// TIA Portal V20 export
FUNCTION_BLOCK "Type_8"   // FB8, GRAPH
// stored: GraphVersion 2.0, SetENOAutomatically false
   // inherited from GRAPH_BASE
   VAR_INPUT
      OFF_SQ { ExternalAccessible := 'False'; ExternalVisible := 'False'; ExternalWritable := 'False'} : Bool := false;   // Turn sequence off
      INIT_SQ { ExternalAccessible := 'False'; ExternalVisible := 'False'; ExternalWritable := 'False'} : Bool := false;   // Set sequence to initial state
      ACK_EF { ExternalAccessible := 'False'; ExternalVisible := 'False'; ExternalWritable := 'False'} : Bool := false;   // Acknowledge all errors and faults
      S_PREV { ExternalAccessible := 'False'; ExternalVisible := 'False'; ExternalWritable := 'False'} : Bool := false;   // Output previous step in parameter S_NO
      S_NEXT { ExternalAccessible := 'False'; ExternalVisible := 'False'; ExternalWritable := 'False'} : Bool := false;   // Indicate next step in parameter S_NO
      SW_AUTO { ExternalAccessible := 'False'; ExternalVisible := 'False'; ExternalWritable := 'False'} : Bool := false;   // Automatic mode
      SW_TAP { ExternalAccessible := 'False'; ExternalVisible := 'False'; ExternalWritable := 'False'} : Bool := false;   // Semiautomatic/switch with transition
      SW_TOP { ExternalAccessible := 'False'; ExternalVisible := 'False'; ExternalWritable := 'False'} : Bool := false;   // Semiautomatic/ignore transition
      SW_MAN { ExternalAccessible := 'False'; ExternalVisible := 'False'; ExternalWritable := 'False'} : Bool := false;   // Manual mode
      S_SEL { ExternalAccessible := 'False'; ExternalVisible := 'False'; ExternalWritable := 'False'} : Int := 0;   // Select step to be output to S_NO
      S_ON { ExternalAccessible := 'False'; ExternalVisible := 'False'; ExternalWritable := 'False'} : Bool := false;   // Activate step indicated in S_NO
      S_OFF { ExternalAccessible := 'False'; ExternalVisible := 'False'; ExternalWritable := 'False'} : Bool := false;   // Disable step indicated in S_NO
      T_PUSH { ExternalAccessible := 'False'; ExternalVisible := 'False'; ExternalWritable := 'False'} : Bool := false;   // Enable transition to switch in semi automatic mode
   END_VAR
   VAR_OUTPUT
      S_NO { ExternalAccessible := 'False'; ExternalVisible := 'False'; ExternalWritable := 'False'} : Int := 0;   // Step number
      S_MORE { ExternalAccessible := 'False'; ExternalVisible := 'False'; ExternalWritable := 'False'} : Bool := false;   // More steps are available and can be shown in S_NO
      S_ACTIVE { ExternalAccessible := 'False'; ExternalVisible := 'False'; ExternalWritable := 'False'} : Bool := false;   // Step indicated in S_NO is active
      ERR_FLT { ExternalAccessible := 'False'; ExternalVisible := 'False'; ExternalWritable := 'False'} : Bool := false;   // Interlock or supervision group error
      AUTO_ON { ExternalAccessible := 'False'; ExternalVisible := 'False'; ExternalWritable := 'False'} : Bool := false;   // Automatic mode is active
      TAP_ON { ExternalAccessible := 'False'; ExternalVisible := 'False'; ExternalWritable := 'False'} : Bool := false;   // Semiautomatic mode/step with transition enabled
      TOP_ON { ExternalAccessible := 'False'; ExternalVisible := 'False'; ExternalWritable := 'False'} : Bool := false;   // Semiautomatic mode/ignore transition enabled
      MAN_ON { ExternalAccessible := 'False'; ExternalVisible := 'False'; ExternalWritable := 'False'} : Bool := false;   // Manual mode is active
   END_VAR
BEGIN
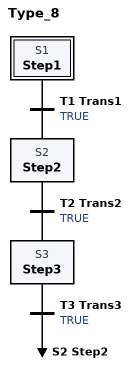
   // sequencer 1
   INITIAL_STEP Step1:   // S1, max time T#10S, warning time T#7S
   END_STEP
   TRANSITION Trans1 FROM Step1 TO Step2   // T1
      := TRUE;
   END_TRANSITION
   STEP Step2:   // S2, max time T#10S, warning time T#7S
   END_STEP
   TRANSITION Trans2 FROM Step2 TO Step3   // T2
      := TRUE;
   END_TRANSITION
   STEP Step3:   // S3, max time T#10S, warning time T#7S
   END_STEP
   TRANSITION Trans3 FROM Step3 TO Step2   // T3, jump
      := TRUE;
   END_TRANSITION
END_FUNCTION_BLOCK
